{attribute 'qualified_only'}
VAR_GLOBAL
END_VAR

(* stored: Version 1.1.0.1, ProductVersion 3.1.4024.12
   GVL gvlHMI: Id {1a90970f-9fe3-4704-bc53-ecbc2633db0d} *)
